Staubli VAL3: SettingGEN.pjx

Parameters version=s7.6 stackSize=5000 millimeterUnit=true
Program file=getErrorMessage.pgx
Program file=Init.pgx
Program file=listFilling.pgx
Program file=readMe.pgx
Program file=start.pgx
Program file=stop.pgx
Data file=SettingGEN.dtx
Library alias=ut path=Disk://Tracking/Tools/util/util.pjx
